{attribute addProperty BoxType "EK1960-2600-0021"}
{attribute addProperty Id "FSOEAT %I*FSOE_3B47B0C112015"}
{attribute addProperty CRC "3417382692"}
{attribute addProperty SizeInBites "120"}
{attribute addProperty SizeInBytes "15"}
TYPE FSoE_Inputs_CBB11F24 :
STRUCT
	{attribute addProperty Name "FSOE"}
	FSOE AT %I* : FSOE_3B47B0C1;
END_STRUCT
END_TYPE

(* stored: Version 1.2.0.0, ProductVersion 3.1.4024.9
   DUT FSoE_Inputs_CBB11F24: Id {f96c08a4-25f1-4c6d-a10b-c302ae50650b} *)
